// TIA Portal V21 export
TYPE "Shift_Register_Data"
   STRUCT
      x_Presence : Bool;
   END_STRUCT;
END_TYPE
